FUNCTION_BLOCK BlockerCtrl (* Template for an empty basic function block *)
  (* Standard: 61499-2 *)
  (* Version 1.0, 2018-09-13, az *)
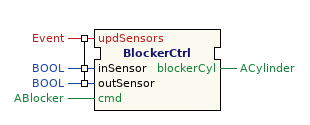
  EVENT_INPUT
    updSensors WITH inSensor, outSensor;
  END_EVENT
  VAR_INPUT
    inSensor : BOOL;
    outSensor : BOOL;
  END_VAR
  SOCKETS
    cmd : ABlocker;
  END_SOCKETS
  PLUGS
    blockerCyl : ACylinder;
  END_PLUGS
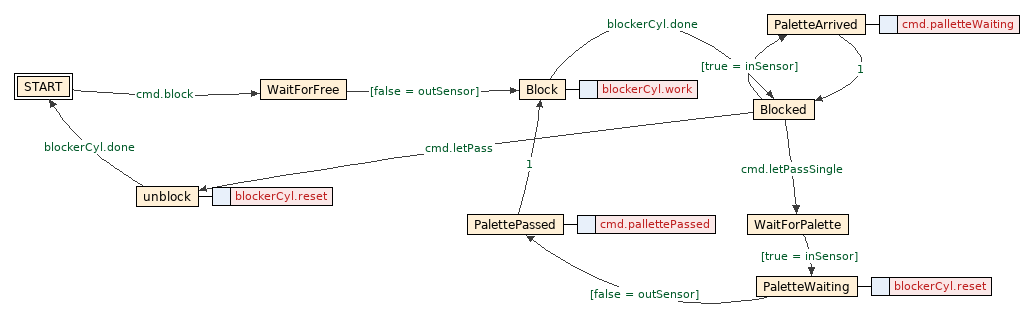
  EC_STATES
    START; (* Initial State *)
    WaitForFree;
    Block : -> blockerCyl.work;
    Blocked;
    PaletteArrived : -> cmd.palletteWaiting;
    WaitForPalette;
    PaletteWaiting : -> blockerCyl.reset;
    PalettePassed : -> cmd.pallettePassed;
    unblock : -> blockerCyl.reset;
  END_STATES
  EC_TRANSITIONS
    START TO WaitForFree := cmd.block;
    WaitForFree TO Block := [false = outSensor];
    Block TO Blocked := blockerCyl.done;
    Blocked TO PaletteArrived := [true = inSensor];
    PaletteArrived TO Blocked := 1;
    Blocked TO WaitForPalette := cmd.letPassSingle;
    WaitForPalette TO PaletteWaiting := [true = inSensor];
    PaletteWaiting TO PalettePassed := [false = outSensor];
    PalettePassed TO Block := 1;
    Blocked TO unblock := cmd.letPass;
    unblock TO START := blockerCyl.done;
  END_TRANSITIONS
END_FUNCTION_BLOCK
